TEXTLIST TextList_UVLed_errorid
  0 = 'no_error'
  1 = 'not_connected'
  2 = 'invalid_state'
  3 = 'unknown_error'
  666 = 'emergency_error'
   = ''
END_TEXTLIST

(* stored: Version 1.1.0.1, ProductVersion 3.1.4024.11
   TextList TextList_UVLed_errorid: Id {35e90247-d389-46d1-9a3a-36e977187aec} *)
